FUNCTION_BLOCK SERVER_22 (* 22 RD/RD Server Interface *)
  (* Standard: 61499-1; Classification: Communications *)
  (* Version 1.0, 2019-07-08, Jose Cabral, fortiss GmbH *)
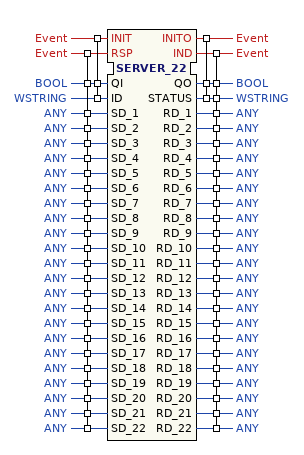
  EVENT_INPUT
    INIT WITH QI, ID;
    RSP WITH QI, SD_1, SD_2, SD_3, SD_4, SD_5, SD_6, SD_7, SD_8, SD_9, SD_10, SD_11, SD_12, SD_13, SD_14, SD_15, SD_16, SD_17, SD_18, SD_19, SD_20, SD_21, SD_22;
  END_EVENT
  EVENT_OUTPUT
    INITO WITH QO, STATUS;
    IND WITH QO, STATUS, RD_1, RD_2, RD_3, RD_4, RD_5, RD_6, RD_7, RD_8, RD_9, RD_10, RD_11, RD_12, RD_13, RD_14, RD_15, RD_16, RD_17, RD_18, RD_19, RD_20, RD_21, RD_22;
  END_EVENT
  VAR_INPUT
    QI : BOOL;
    ID : WSTRING;
    SD_1 : ANY; (* Data to Send *)
    SD_2 : ANY; (* Data to Send *)
    SD_3 : ANY; (* Data to Send *)
    SD_4 : ANY; (* Data to Send *)
    SD_5 : ANY; (* Data to Send *)
    SD_6 : ANY; (* Data to Send *)
    SD_7 : ANY; (* Data to Send *)
    SD_8 : ANY; (* Data to Send *)
    SD_9 : ANY; (* Data to Send *)
    SD_10 : ANY; (* Data to Send *)
    SD_11 : ANY; (* Data to Send *)
    SD_12 : ANY; (* Data to Send *)
    SD_13 : ANY; (* Data to Send *)
    SD_14 : ANY; (* Data to Send *)
    SD_15 : ANY; (* Data to Send *)
    SD_16 : ANY; (* Data to Send *)
    SD_17 : ANY; (* Data to Send *)
    SD_18 : ANY; (* Data to Send *)
    SD_19 : ANY; (* Data to Send *)
    SD_20 : ANY; (* Data to Send *)
    SD_21 : ANY; (* Data to Send *)
    SD_22 : ANY; (* Data to Send *)
  END_VAR
  VAR_OUTPUT
    QO : BOOL;
    STATUS : WSTRING;
    RD_1 : ANY; (* Received Data *)
    RD_2 : ANY; (* Received Data *)
    RD_3 : ANY; (* Received Data *)
    RD_4 : ANY; (* Received Data *)
    RD_5 : ANY; (* Received Data *)
    RD_6 : ANY; (* Received Data *)
    RD_7 : ANY; (* Received Data *)
    RD_8 : ANY; (* Received Data *)
    RD_9 : ANY; (* Received Data *)
    RD_10 : ANY; (* Received Data *)
    RD_11 : ANY; (* Received Data *)
    RD_12 : ANY; (* Received Data *)
    RD_13 : ANY; (* Received Data *)
    RD_14 : ANY; (* Received Data *)
    RD_15 : ANY; (* Received Data *)
    RD_16 : ANY; (* Received Data *)
    RD_17 : ANY; (* Received Data *)
    RD_18 : ANY; (* Received Data *)
    RD_19 : ANY; (* Received Data *)
    RD_20 : ANY; (* Received Data *)
    RD_21 : ANY; (* Received Data *)
    RD_22 : ANY; (* Received Data *)
  END_VAR
END_FUNCTION_BLOCK
